TYPE Stoffwerte :
STRUCT
	Temperatur 	: REAL; //°C
	Dichte		: REAL; //kg/m³
	Cp			: REAL;	//kJ/kg K
END_STRUCT
END_TYPE

(* stored: Version 1.1.0.1, ProductVersion 3.1.4018.5
   DUT Stoffwerte: Id {a9d357f2-ecb0-4c75-9d71-911c2b7f6b34} *)
